Fanuc TP program (LS listing): STRF_SELECT.LS

/PROG  STRF_SELECT
/ATTR
OWNER		= MNEDITOR;
COMMENT		= "string probe";
PROG_SIZE	= 0;
CREATE		= DATE 26-01-01  TIME 00:00:00;
MODIFIED	= DATE 26-01-01  TIME 00:00:00;
FILE_NAME	= ;
VERSION		= 0;
LINE_COUNT	= 3;
MEMORY_SIZE	= 0;
PROTECT		= READ_WRITE;
TCD:  STACK_SIZE	= 0,
      TASK_PRIORITY	= 50,
      TIME_SLICE	= 0,
      BUSY_LAMP_OFF	= 0,
      ABORT_REQUEST	= 0,
      PAUSE_REQUEST	= 0;
DEFAULT_GROUP	= 1,*,*,*,*;
CONTROL_CODE	= 00000000 00000000;
/MN
   1:  SELECT SR[20]='A',JMP LBL[1] ;
   2:         ELSE,JMP LBL[1] ;
   3:  LBL[1] ;
/POS
/END
